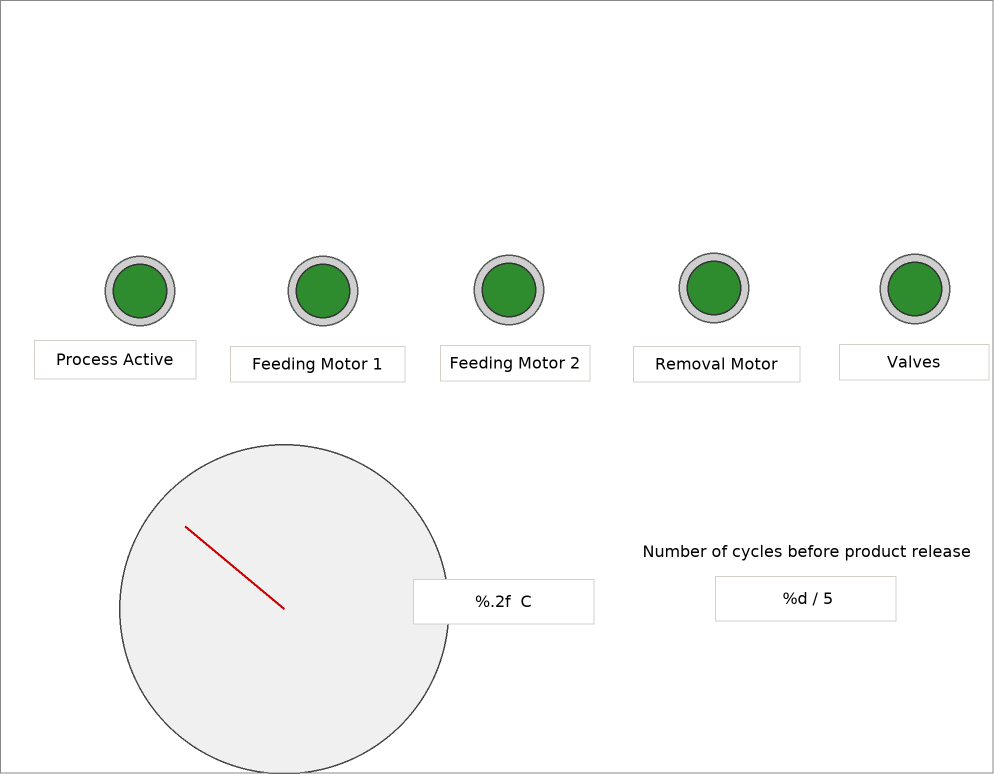
VISUALIZATION Visualization  // 994x774, background image ImagePool.Keskisuuri+600px(näytöille,+RGB,+JPG)+HAMK_HAMK_Logo_text_large_FIN
    Textfield (34,340 162x39), "Process Active"
    Lamp1 (97,250 86x82), variable: drive.bProcessActive, style: Lamp-Lamp1-Green
    Lamp1 (280,250 86x82), variable: drive.bM1active, style: Lamp-Lamp1-Green
    Lamp1 (466,249 86x82), variable: drive.bFeedMotor2Lamp, style: Lamp-Lamp1-Green
    Lamp1 (671,247 86x82), variable: drive.bM2active, style: Lamp-Lamp1-Green
    Textfield (230,346 175x36), "Feeding Motor 1"
    Textfield (440,345 150x36), "Feeding Motor 2"
    Textfield (633,346 167x36), "Removal Motor"
    Meter360 (33,444 502x330), value: drive.ScaledThermoCouple2Value, style: Meter-Meter360-Yellow, scale format: %.1f, scale 0..800
    Lamp1 (872,248 86x82), variable: drive.bValveLamp, style: Lamp-Lamp1-Green
    Textfield (839,344 150x36), "Valves"
    Textfield (413,579 181x45), "%.2f C", text variable: drive.ScaledThermoCouple2Value
    Textfield (715,576 181x45), "%d / 5", text variable: drive.itopvalvecount
    Label (620,519 374x65), "Number of cycles before product release"
END_VISUALIZATION

(* stored: Version 1.1.0.1, ProductVersion 3.1.4024.12
   Visu Visualization: Id {1634d76f-269e-4291-9a0e-eb7c5ac94af6} *)
